TYPE U_EMS_HS_Write :
UNION
	aWords					: ARRAY [1..8] OF WORD;
	stVars					: ST_EMS_HS_Write;

END_UNION
END_TYPE

(* stored: Version 1.1.0.1, ProductVersion 3.1.4024.2
   DUT U_EMS_HS_Write: Id {85a1e226-7f8f-41bb-b4a5-ac16c19541ec} *)
